Fanuc KAREL source: DEL_INST_TPE.kl

PROGRAM T
%NOLOCKGROUP
VAR
 v0 : INTEGER
 v1 : INTEGER
 v2 : INTEGER
BEGIN
 DEL_INST_TPE(v0, v1, v2)
END T
